# B&R Automation Studio project ksuTCPExample
Automation Studio 4.9

## Configuration Config1

CPU X20CP1586, AutomationRuntime C4.92, Build 4.1.2, Vc V4.72.5

### Task classes (Cpu.sw)
```
Cyclic#8:
  Client <- TCPComms.Client.prg
  Server <- TCPComms.Server.prg [disabled]
Libraries: AsTCP, runtime, BRSE_JSON, astime, sys_lib, AsBrStr, standard, asstring, Queue
```

### Hardware
```
X20CP1586 : X20CP1586 v1.10.0.0
  Connector IF2:
    ActivateDevice = 1
  ConfigurationID = ksuTCPExample_Config1
  Simulation = 1
  VolatileGlobalPvSize = 210000
  FileDevice1
  FileDeviceName1 = USER
  FileDevicePath1 = USER_PATH
```

## Logical view

Binary libraries used (declarations not repeated): operator, runtime, astime, AsIecCon, AsTCP, sys_lib, AsBrStr, standard, asstring

### Global.typ - Global data types
```iecst
TYPE
	MessageToEZ3_typ : 	STRUCT
		Move_Command : STRING[20];
		Parameter_One : STRING[20];
		Parameter_Two : STRING[20];
		Battery_Subscribe : BOOL;
	END_STRUCT;
END_TYPE
```

### Global.var - Global variables
```iecst
VAR
	gSendQueue : FifoQueue_typ;
	gMessageToEZ3 : MessageToEZ3_typ;
END_VAR
```

### Package Logical/Libraries - Global libraries

### Library Logical/Libraries/BRSE_JSON (ANSIC, version 1.00.1) - A new source library
Depends on: sys_lib, astime, AsBrStr

#### BRSE_JSON.fun - Exported functions and function blocks
```iecst
(********************************************************************
 * COPYRIGHT -- B&R
 ********************************************************************
 * Library: Library
 * File: Library.fun
 * Author: Florian Damerow
 * Created: March 09, 2011
 ********************************************************************
 * Functions and function blocks of library Library
 ********************************************************************)

FUNCTION_BLOCK JSON_Parse (*parses a JSON message and writes the content to the structure on the PLC*)
	VAR_INPUT
		pMessage : REFERENCE TO UDINT; (*Pointer to the JSON Message (String)*)
		pDebug : REFERENCE TO UDINT; (*Pointer Debug Buffer (String)*)
		pVariablesNotFound : REFERENCE TO UDINT; (*Pointer Buffer of VariablesNotFound (String)*)
		SizeVariablesNotFound : UDINT; (*size of the VariablesNotFound Buffer*)
		SizeDebug : UDINT; (*size of the Debug Buffer*)
	END_VAR
	VAR_OUTPUT
		ErrorInfo : UINT;
	END_VAR
	VAR
		parselevel : USINT;
		pvIndex : ARRAY[0..MAX_STRUCT_DEPTH_Parse] OF INT;
		Buffer : STRING[80];
		parsestateold : USINT;
		parsestate : USINT;
		pvName : ARRAY[0..MAX_STRUCT_DEPTH_Parse] OF STRING[64];
		isArray : ARRAY[0..MAX_STRUCT_DEPTH_Parse] OF BOOL;
		fullName : STRING[MAX_STRUCT_NAME_LENGTH_Parse];
		j : UINT;
	END_VAR
END_FUNCTION_BLOCK

FUNCTION_BLOCK JSON_Stringify (*converts a PV variable and the whole structure into a JSON Object using PV_ninfo*)
	VAR_INPUT
		pStName : REFERENCE TO UDINT; (*address to variable name (STRING)*)
	END_VAR
	VAR_OUTPUT
		Status : UINT; (*address to status-variable 0=not done; 1=done; 2=error*)
		Output : STRING[MAX_OUTPUT_LENGTH_Stringify]; (*Output contains the content of one step*)
	END_VAR
	VAR
		tmpStruct : STRING[MAX_OUTPUT_LENGTH_Stringify];
		pvName : ARRAY[0..MAX_STRUCT_DEPTH_Stringify] OF STRING[100];
		j : UDINT;
		pvIndex : ARRAY[0..MAX_STRUCT_DEPTH_Stringify] OF UINT;
		TaskDoc : TaskDoc1_typ;
		pvType : UDINT;
		pvLength : UDINT;
		arrMem : ARRAY[0..MAX_STRUCT_DEPTH_Stringify] OF UINT;
		pvStructMembers : ARRAY[0..MAX_STRUCT_DEPTH_Stringify] OF UINT;
		tmpValue : STRING[MAX_OUTPUT_LENGTH_Stringify];
		Buffer : STRING[MAX_OUTPUT_LENGTH_Stringify];
		i : DINT;
		pvLevel : DINT;
		tmpDepth : STRING[MAX_OUTPUT_LENGTH_Stringify];
		state : USINT;
		pvContinue : BOOL;
		pvSearchComplete : BOOL;
		data_len : UDINT;
		isArray : ARRAY[0..MAX_STRUCT_DEPTH_Stringify] OF BOOL;
		arrIndex : UINT;
		pv_adresse : UDINT;
	END_VAR
END_FUNCTION_BLOCK
```

#### BRSE_JSON.c
```c
/*! \file BRSE_JSON.c */
/********************************************************************
 * COPYRIGHT -- B&R
 ********************************************************************
 * Library: BRSE_JSON
 * File: BRSE_JSON.c
 * Author: Florian Damerow
 * Created: March 09, 2011
 *******************************************************************/

#include <bur/plctypes.h>
#include "BRSE_JSON.h"
#include <AsBrStr.h>
#include <string.h>
#include "BRSE_JSON_Main.h"
STRING tmpVal[80];

UDINT ValToString(UDINT pv_adresse, UINT pvType){
	switch (pvType) {
		case 1: {
				BOOL *var = (BOOL *)pv_adresse;
				brsitoa((BOOL)*var,(UDINT)&tmpVal);
				break;
				}
		case 2: {
				SINT *var = (SINT *)pv_adresse;
				brsitoa((SINT)*var,(UDINT)&tmpVal);
				break;
				}
		case 3: {
				INT *var = (INT *)pv_adresse;
				brsitoa((INT)*var,(UDINT)&tmpVal);
				break;
				}
		case 4: {
				DINT *var = (DINT *)pv_adresse;
				brsitoa((DINT)*var,(UDINT)&tmpVal);
				break;
				}
		case 5: {
				USINT *var = (USINT *)pv_adresse;
				brsitoa((USINT)*var,(UDINT)&tmpVal);
				break;
				}
		case 6: {
				UINT *var = (UINT *)pv_adresse;
				brsitoa((UINT)*var,(UDINT)&tmpVal);
				break;
				}
		case 7: {
				UDINT *var = (UDINT *)pv_adresse;
				brsitoa((UDINT)*var,(UDINT)&tmpVal);
				break;
				}
		case 8: {
				REAL *var = (REAL *)pv_adresse;
				brsftoa((REAL)*var,(UDINT)&tmpVal);
				break;
				}
		case 9: {
				STRING *var = (STRING *)pv_adresse;
				STRING *tmpBuffer = (STRING *)&tmpVal;
				strcpy(tmpVal,"\"");
				tmpBuffer++;
				strncpy(tmpBuffer,var,(sizeof(tmpVal)-3));
				strcat(tmpVal,"\"");
				break;
				}
		case 11:{
				DINT *var = (DINT *)pv_adresse;
				STRING *tmpBuffer = (STRING *)&tmpVal;
				strcpy(tmpVal,"\"");
				tmpBuffer++;
				brsitoa((DINT)*var,(UDINT)tmpBuffer);
				strcat(tmpVal,"\"");
				break;
				}
		case 12:{
				DINT *var = (DINT *)pv_adresse;
				STRING *tmpBuffer = (STRING *)&tmpVal;
				strcpy(tmpVal,"\"");
				tmpBuffer++;
				brsitoa((DINT)*var,(UDINT)tmpBuffer);
				strcat(tmpVal,"\"");
				break;
				}
		case 14:{
				LREAL *var = (LREAL *)pv_adresse;
				brsftoa((LREAL)*var,(UDINT)&tmpVal);
				break;
			}
		/*case 11:{
				TIME *var = pv_adresse;
				STRING *ptmpValue = &tmpValue;
				strcpy(ptmpValue,"\\/Date(");
				ptmpValue = ptmpValue + 7;
				itoa((DINT)*var,ptmpValue);
				strcat(ptmpValue,")\\/");
				break;
				}
		case 11:{
				DATE_AND_TIME *var = pv_adresse;
				BRSE_DTF_DateTimeFormat_typ format;
				UDINT error;
				error = BRSE_DTF_CreateFormat("YYYY-MM-DD-hh:mm:ss", &format);
				if(error == 0){
					BRSE_DTF_DTToString((DATE_AND_TIME)*var, &format, tmpValue);
				}
				break;
				}
		case 12:{
				TIME *var = pv_adresse;
				STRING *ptmpValue = &tmpValue;
				strcpy(ptmpValue,"\\/Time(");
				ptmpValue = ptmpValue + 7;
				itoa((DINT)*var,ptmpValue);
				strcat(ptmpValue,")\\/");
				break;
				}*/
		default: strcpy(tmpVal,"null");
				 break;
	}
	return (UDINT)tmpVal;
}

/*! \interface JSON_Parse
	\brief parses a JSON message and writes the content to the structure on the PLC

	This function block parses the JSON message and writes the content to the structure on the PLC using PV_xgetadr.\n
	The structure must exist.\n
	\n
	It is possible to parse a long JSON message in several pieces. The message can be split at every point.\n
	It is only possible to parse JSON Objects '{name:content}' \n
	arrays or non objects are NOT supported e.g. '[name:content, name2:content2]' or 'name:content' \n
	\n
	The maximal possible struture name is defined in MAX_STRUCT_NAME_LENGTH_Parse. \n
	That means the whole name e.g. 'Structure.Outer[1].Inner.Test' is limited. \n
	\n
	Entering an object will result in going up with the level by 1 \n
	Entering an array will result in going up with the level by 1 \n
	Entering an struct array will result in going up with the level by 2 \n
	\n
	If pDebug != 0 the whole message will be written there. This will be done with the state for every character.\n
	If pDebug = 0 no Debugging will be performed by the system.\n

	If pVariablesNotFound != 0 all Variables found in the Message, but could not be written on the system are listed here.
	They are represented in a JSON array e.g. '["var1","var2"]'.\n
	If pVariablesNotFound = 0 no output will performed wen variables could not be written.\n
	\n
	The funktion block will be stopped when an error accured.\n
	The function block will not be stopped when a warning accures.\n
	\par Errors:\n
	\arg 1001	invalid JSON in parsestate 0
	\arg 1002	invalid JSON in parsestate 1
	\arg 1003	invalid JSON in parsestate 3
	\arg 1004	invalid JSON in parsestate 4
	\arg 1005	invalid JSON in parsestate 6
	\arg 1006	invalid JSON in parsestate 7
	\arg 1007	Structure depth is deeper than MAX_STRUCT_DEPTH_Parse

	\par Warnings:\n
	\arg 3001	data type not supported
	\arg 3002	variable not found

	\par General: \n
	\arg 2001	parsing so far successful, but end of JSON message net reached yet
	\arg 0		successfuly finished parsing

	\param[in] pMessage Pointer to the JSON Message (String)
	\param[in] pDebug Pointer Debug Buffer (String)
	\param[in] SizeDebug size of the Debug Buffer
	\param[in] pVariablesNotFound Pointer Buffer of VariablesNotFound (String)
	\param[in] SizeVariablesNotFound size of the VariablesNotFound Buffer

	\param[out] ErrorInfo contains the Error/Warning/General Codes.

*/

void JSON_Parse(struct JSON_Parse* inst)
{
	STRING *message = (STRING *)inst->pMessage;
	STRING *pBuff = (STRING *)inst->pMessage;
	UDINT pBuffOld = 0;
	inst->ErrorInfo = 0;
	while((UDINT)pBuff<((UDINT)message+strlen(message)) && (inst->ErrorInfo < 1000 || inst->ErrorInfo >=2000)){
		switch(inst->parsestate){
			case 0:
				if(*pBuff == '{'){
					inst->parsestate = 1;
					inst->parselevel++;
					pBuff++;
					if(inst->pVariablesNotFound != 0 && inst->SizeVariablesNotFound > 2){
						strcpy((STRING *)inst->pVariablesNotFound,"[");
					}
				}
				else if(*pBuff == ' '){
					pBuff++;
				}
				else{
					inst->ErrorInfo = 1001; /*invalid JSON*/
					return;
				}
				break;

			case 1:
				if(*pBuff == '"'){
					inst->parsestate = 2;
					pBuff++;
				}
				else if(*pBuff == ' '){
					pBuff++;
				}
				else{
					inst->ErrorInfo = 1002; /*invalid JSON*/
					return;
				}
				break;

			case 2:
				if(*pBuff != '"'){
					inst->pvName[inst->parselevel][inst->j] = *pBuff;
					inst->j++;
					pBuff++;
				}
				else {
					inst->pvName[inst->parselevel][inst->j] = '\0';
					inst->j = 0;
					inst->parsestate = 3;
					pBuff++;
				}
				break;

			case 3:
				if(*pBuff == ':'){
					inst->parsestate = 4;
					pBuff++;
				}
				else if(*pBuff == ' '){
					pBuff++;
				}
				else{
					inst->ErrorInfo = 1003; /*invalid JSON*/
					return;
				}
				break;

			case 4:
				if(*pBuff == '{'){
					inst->parsestate = 1;
					inst->parselevel++;
					pBuff++;
				}
				else if(*pBuff == '['){
					/*strcat(inst->pvName[inst->parselevel],"[");
					strcat(inst->pvName[inst->parselevel],"0");
					strcat(inst->pvName[inst->parselevel],"]");*/
					inst->isArray[inst->parselevel] = 1;
					inst->parselevel++;
					pBuff++;
				}
				else if(*pBuff == '\"'){
					inst->Buffer[inst->j] = *pBuff;
					pBuff++;
					inst->j++;
					inst->parsestate = 41;
				}
				else if(*pBuff != '{' && *pBuff != ' ' && *pBuff != '['){ /*maybe better to check for " or - or number*/
					inst->parsestate = 5;
				}
				else if(*pBuff == ' '){
					pBuff++;
				}
				else{
					inst->ErrorInfo = 1004; /*invalid JSON*/
					return;
				}
				break;

			case 41: /* is in String */
				if(*pBuff == '\"'){
					inst->Buffer[inst->j] = *pBuff;
					inst->j++;
					inst->Buffer[inst->j] = '\0';
					inst->j=0;
					pBuff++;
					inst->parsestate = 51;
				}
				else if(*pBuff == '\\'){
					inst->Buffer[inst->j] = *pBuff;
					inst->j++;
					pBuff++;
					inst->Buffer[inst->j] = *pBuff;
					inst->j++;
					pBuff++;
				}
				else{
					inst->Buffer[inst->j] = *pBuff;
					inst->j++;
					pBuff++;
				}
				break;

			case 5:
				if(*pBuff != '}' && *pBuff != ' ' && *pBuff != ',' && *pBuff != ']'){
					inst->Buffer[inst->j] = *pBuff;
					inst->j++;
					pBuff++;
				}
				else{
					inst->Buffer[inst->j] = '\0';
					inst->j=0;
					inst->parsestate = 51;
				}
				break;

			case 51: /*write variable*/
				memset((UDINT *)(inst->fullName),0,sizeof(inst->fullName));
				{
					UINT i = 1;
					UDINT adresse;
					UDINT datalen;
					UDINT pvType;
					UDINT pvLength;
					UINT pvStructMembers;
					STRING tmpStr[5];
					while(i <= inst->parselevel && (sizeof(inst->fullName)-strlen(inst->fullName)-7) > strlen(inst->pvName[i])){
						strcat(inst->fullName,inst->pvName[i]);
						if(inst->isArray[i] == 1){
							strcat(inst->fullName,"[");
							brsitoa(inst->pvIndex[i],(UDINT)&tmpStr);
							strcat(inst->fullName,tmpStr);
							strcat(inst->fullName,"]");
						}
						if(i < inst->parselevel && inst->isArray[i] == 0){
							strcat(inst->fullName,".");
						}
						i++;
					}
					inst->ErrorInfo = PV_ninfo((STRING *)&inst->fullName, &pvType, &pvLength, &pvStructMembers);
					if(inst->ErrorInfo == 0){
						inst->ErrorInfo = PV_xgetadr((STRING *)&inst->fullName, &adresse, &datalen);
					}
					else{
						inst->ErrorInfo = 3002; /* variable not found */
					}
					if(inst->ErrorInfo == 0){
						STRING *Buffer = (STRING *)&inst->Buffer;
						if(*Buffer == '\"'){
							Buffer++;
							if(inst->Buffer[strlen(Buffer)] == '\"'){
								inst->Buffer[strlen(Buffer)] = '\0';
							}
						}
						if(strstr(inst->Buffer,"null") == 0){
							switch(pvType){
								case 0:{
									DINT *adr = (DINT *)adresse;
									*adr = (DINT)brsatoi((UDINT)Buffer);
									break;
									}
								case 1:{
									BOOL *adr = (BOOL *)adresse;
									if(brsatoi((UDINT)Buffer) != 0){
										*adr = 1;
									}
									else{
										*adr = 0;
									}
									break;
									}
								case 2:{
									SINT *adr = (SINT *)adresse;
									*adr = (SINT)brsatoi((UDINT)Buffer);
									break;
									}
								case 3:{
									INT *adr = (INT *)adresse;
									*adr = (INT)brsatoi((UDINT)Buffer);
									break;
									}
								case 4:{
									DINT *adr = (DINT *)adresse;
									*adr = (DINT)brsatoi((UDINT)Buffer);
									break;
									}
								case 5:{
									USINT *adr = (USINT *)adresse;
									*adr = (USINT)brsatoi((UDINT)Buffer);
									break;
									}
								case 6:{
									UINT *adr = (UINT *)adresse;
									*adr = (UINT)brsatoi((UDINT)Buffer);
									break;
									}
								case 7:{
									UDINT *adr = (UDINT *)adresse;
									*adr = (UDINT)brsatoi((UDINT)Buffer);
									break;
									}
								case 8:{
									REAL *adr = (REAL *)adresse;
									*adr = (REAL)brsatof((UDINT)Buffer);
									break;
									}
								case 9:{
									STRING *adr = (STRING *)adresse;
									strncpy(adr, Buffer, pvLength-1);
									break;
									}
								case 11:{
									DINT *adr = (DINT *)adresse;
									*adr = (DINT)brsatoi((UDINT)Buffer);
									break;
									}
								case 12:{
									DINT *adr = (DINT *)adresse;
									*adr = (DINT)brsatoi((UDINT)Buffer);
									break;
									}
								case 14:{
										LREAL *adr = (LREAL *)adresse;
										*adr = (LREAL)brsatof((UDINT)Buffer);
										break;
									}
								/*case 11:{
									DINT *adr = adresse;
									STRING *Buffer = &inst->Buffer;
									Buffer = strstr(inst->Buffer,")\\/");
									if(Buffer != 0){
										*Buffer = '\0';
										Buffer = strstr(inst->Buffer,"\\/Date(");
										if(Buffer != 0){
											Buffer = Buffer + 7;
										}
									}
									*adr = (DINT)atoi(Buffer);
									break;
									}
								case 12:{
									DINT *adr = adresse;
									STRING *Buffer = &inst->Buffer;
									Buffer = strstr(inst->Buffer,")\\/");
									if(Buffer != 0){
										*Buffer = '\0';
										Buffer = strstr(inst->Buffer,"\\/Time(");
										if(Buffer != 0){
											Buffer = Buffer + 7;
										}
									}
									*adr = (DINT)atoi(Buffer);
									break;
									}*/

								default:{
									inst->ErrorInfo = 3001;
									break;
									}
							}
						}
					}
					else{
						inst->ErrorInfo = 3002; /* variable not found */
						if(inst->pVariablesNotFound != 0 && inst->SizeVariablesNotFound != 0){
							if((inst->SizeVariablesNotFound - strlen((STRING *)inst->pVariablesNotFound)-2) > strlen(inst->fullName)+3){
								if(strlen((STRING *)inst->pVariablesNotFound) > 2){
									strcat((STRING *)inst->pVariablesNotFound,",");
								}
								strcat((STRING *)inst->pVariablesNotFound,"\"");
								strcat((STRING *)inst->pVariablesNotFound,inst->fullName);
								strcat((STRING *)inst->pVariablesNotFound,"\"");
							}
						}
					}
					if(*pBuff == ',' && inst->isArray[inst->parselevel-1] == 1){
						pBuff++;
						inst->pvIndex[inst->parselevel-1]++;
						inst->parsestate = 4;
					}
					else{
						inst->parsestate = 6;
					}
				}
				break;

			case 6:
				if(*pBuff == '}'){
					inst->parsestate = 6;
					inst->pvIndex[inst->parselevel-1] = 0;
					inst->parselevel--;
					pBuff++;
				}
				else if(*pBuff == ']'){
					inst->parsestate = 6;
					inst->pvIndex[inst->parselevel-1] = 0;
					inst->parselevel--;
					inst->isArray[inst->parselevel] = 0;
					pBuff++;
				}
				else if(*pBuff == ','){
					inst->parsestate = 7;
					inst->pvIndex[inst->parselevel-1]++;
					pBuff++;
				}
				else if(*pBuff == ' '){
					pBuff++;
				}
				else{
					inst->ErrorInfo = 1005; /*invalid JSON*/
					return;
				}
				break;

			case 7:
				if(*pBuff == '{'){
					inst->parselevel++;
					inst->parsestate = 1;
					pBuff++;
				}
				else if(*pBuff == '\"'){
					inst->parsestate = 1;
				}
				else if(*pBuff == ' '){
					pBuff++;
				}
				else{
					inst->ErrorInfo = 1006; /*invalid JSON*/
					return;
				}
		}

		/* DEBUGGING */
		if(inst->pDebug != 0){
			if(pBuffOld != (UDINT)pBuff){
				STRING BUFFER2[4];
				STRING BUFFER3[2];
				if((inst->SizeDebug - strlen((STRING *)inst->pDebug) - 1) > 7){
					if(inst->parsestateold != inst->parsestate){
						inst->parsestateold = inst->parsestate;
						brsitoa((DINT)inst->parsestate,(UDINT)&BUFFER2);
						strcat((STRING *)inst->pDebug,"(");
						strcat((STRING *)inst->pDebug,BUFFER2);
						strcat((STRING *)inst->pDebug,")");
					}
					BUFFER3[0] = *pBuff;
					BUFFER3[1] = 0;
					strcat((STRING *)inst->pDebug,BUFFER3);
				}
			}
			pBuffOld = (UDINT)pBuff;
		}
	}
	/* Error Handling */
	if(inst->parselevel > MAX_STRUCT_DEPTH_Parse){
		inst->ErrorInfo = 1007;
	}
	if(inst->ErrorInfo >= 1000 && inst->ErrorInfo  < 2000){
		inst->parselevel = 0;
		inst->parsestate = 0;
		memset(inst->pvIndex,0,sizeof(inst->pvIndex));
		memset(inst->pvName,0,sizeof(inst->pvName));
	}
	else if(inst->parselevel != 0){
		inst->ErrorInfo = 2001; /*not done*/
	}
	else{
		if(inst->pVariablesNotFound != 0){
			strcat((STRING *)inst->pVariablesNotFound,"]");
		}
		inst->parsestate = 0;
	}
}

/*! \interface JSON_Stringify
	\brief converts a PV variable and the whole structure into a JSON Object using PV_ninfo.

	This function block converts the whole structure of a PV variable into a JSON Object using PV_ninfo. \n
	The variable name should be the same as using the PV_ninfo function. By that it is possible to access any kind of PV variables.\n
	The output is always a JSON object. e.g. '{"varname": ... }' \n
	\n
	The function block has to be run several times until the Status = 1. \n
	Every time the function block is called it creates the JSON output for one new variable inside the Structure. \n
	If the variable in the structure is an array of a non object type the whole array will be created in Output.\n
	\n
	The maximum Output length is defined by MAX_OUTPUT_LENGTH_Stringify.\n
	The maximum Value of a nun array, non structure variable is 80. So Strings are only supported up the 80 characters.\n

	\par Status Codes:\n
	\arg 1001 Variable not found
	\arg 1002 Variable value too long
	\arg 1 singify process completed
	\arg 0 singify process not completet yet - run again

	\param[in] pStName Pointer to the requested variable name

	\param[out] Status returns the Status codes
	\param[out] Output contains the content of one step

*/
void JSON_Stringify(struct JSON_Stringify* inst)
{
	STRING *pBuff = 0;
	STRING strBuff[20];
	inst->TaskDoc.Input.StructDepth = MAX_STRUCT_DEPTH_Stringify;
	/*gather information of the structure item*/
	memset(inst->tmpStruct,0,sizeof(inst->tmpStruct));
	strcpy(inst->tmpStruct,(STRING *)inst->pStName);

	strcat(inst->tmpStruct, inst->pvName[0]);
	for( inst->i = 1; inst->i <= inst->pvLevel; inst->i++ ){
		if(inst->isArray[inst->i-1] == 0){
			strcat(inst->tmpStruct, ".");
			strcat(inst->tmpStruct, inst->pvName[inst->i]);
		}
		else{
			inst->isArray[inst->pvLevel] = 1;
			strcat(inst->tmpStruct,"[");
			brsitoa(inst->pvIndex[inst->i-1],(UDINT)&strBuff);
			strcat(inst->tmpStruct,strBuff);
			strcat(inst->tmpStruct,"]");
		}
	}
	/*Search in PV-list*/
	inst->TaskDoc.Output.StatusInfo = PV_ninfo((STRING *)&inst->tmpStruct, &inst->pvType, &inst->pvLength, &inst->pvStructMembers[inst->pvLevel]);
	if(inst->pvType == 0){
		STRING name[80];
		inst->TaskDoc.Output.StatusSearch = PV_item((STRING *)&inst->tmpStruct, 0, (STRING *)&name);
		if(inst->TaskDoc.Output.StatusSearch != 0){
			inst->pvType = 4;
			inst->pvStructMembers[inst->pvLevel] = 1;
			inst->TaskDoc.Output.StatusSearch = 0;
		}
	}
	if(inst->pvType == 15){
		inst->isArray[inst->pvLevel] = 1;
		strcat(inst->tmpStruct,"[");
		brsitoa(inst->pvIndex[inst->pvLevel],(UDINT)&strBuff);
		strcat(inst->tmpStruct,strBuff);
		strcat(inst->tmpStruct,"]");
		inst->pvLevel = inst->pvLevel + 1;
		inst->TaskDoc.Output.StatusInfo = PV_ninfo((STRING *)&inst->tmpStruct, &inst->pvType, &inst->pvLength, &inst->pvStructMembers[inst->pvLevel]);
	}
	else{
		inst->isArray[inst->pvLevel] = 0;
	}
	if( inst->TaskDoc.Output.StatusInfo == 0 ){
		inst->TaskDoc.Output.StatusInfo = PV_xgetadr((STRING *)&inst->tmpStruct,&inst->pv_adresse,&inst->data_len);
	}
	if( inst->TaskDoc.Output.StatusInfo == 0 ){
	/*variable was found*/
		STRING *ValToStr;
		UDINT Size=0;
		memset(inst->tmpValue,0,sizeof(inst->tmpValue));
		if(inst->pvStructMembers[inst->pvLevel]>1){
			strcat(inst->tmpValue,"[");
		}
		ValToStr = (STRING *)ValToString(inst->pv_adresse, inst->pvType);
		if((sizeof(inst->tmpValue)-strlen(inst->tmpValue)-2) > strlen(ValToStr)){
			strcat(inst->tmpValue, ValToStr);
		}
		inst->arrIndex = 1;
		Size = (UDINT)(inst->data_len/inst->pvStructMembers[inst->pvLevel]);
		pBuff = (STRING *)((UDINT)inst->pv_adresse+Size);
		/*build array output */
		while(inst->arrIndex < inst->pvStructMembers[inst->pvLevel]){
			ValToStr = (STRING *)ValToString((UDINT)pBuff, inst->pvType);
			if((sizeof(inst->tmpValue)-strlen(inst->tmpValue)-2) <= strlen(ValToStr)){
				inst->Status = 1002; /*Variable Value too long*/
				return;
			}
			strcat(inst->tmpValue, ",");
			strcat(inst->tmpValue, ValToStr);
			pBuff = pBuff+Size;
			inst->arrIndex++;
		}
		if(inst->pvStructMembers[inst->pvLevel]>1){
			strcat(inst->tmpValue,"]");
		}

		/*get inner variable name*/
		pBuff = (inst->tmpStruct)+strlen(inst->tmpStruct);
		while((UDINT)pBuff >= (UDINT)&(inst->tmpStruct) && *pBuff != '.'){
			pBuff--;
		}
		pBuff++;
		/*create JSON output*/
		memset(inst->Output,0,sizeof(inst->Output));
		if((43+strlen(inst->tmpValue)) > sizeof(inst->Output)){
			inst->Status = 1002; /*Variable Value too long*/
			return;
		}
		if(!(inst->isArray[inst->pvLevel-1] == 1 && inst->pvIndex[inst->pvLevel-1] > 0)){
			if((inst->pvLevel == 0 && inst->pvIndex[0] == 0) || (inst->isArray[inst->pvLevel-1] == 1 && (inst->pvLevel-1) == 0) ){
				strcat(inst->Output, "{");

			}
			strcat(inst->Output, "\"");
			if( inst->pvLevel == 0){
				strcat(inst->Output, (STRING *)inst->pStName);
			}
			else if(inst->isArray[inst->pvLevel-1] == 1){
				if((inst->pvLevel-1) > 0){
					strcat(inst->Output, inst->pvName[inst->pvLevel-1]);
				}
				else{
					strcat(inst->Output, (STRING *)inst->pStName);
				}
			}else{
				strcat(inst->Output, inst->pvName[inst->pvLevel]);
			}
			strcat(inst->Output, "\":");
			if(inst->isArray[inst->pvLevel-1]){
				strcat(inst->Output, "[");
			}
		}
		if( inst->pvType == 0 ){
			strcat(inst->Output, "{");
		}
		if( inst->pvType != 0 && inst->pvType != 15 ){
			strcat(inst->Output, inst->tmpValue);
		}

		inst->pvSearchComplete = 0;

		if( (inst->pvType == 0) && (inst->pvLevel < (inst->TaskDoc.Input.StructDepth-1)) ){
			/*variable is a structure and its ok to go look inside it*/
			/*ok. proceed to next level.*/
			inst->TaskDoc.Output.StatusSearch = PV_item((STRING *)&inst->tmpStruct, inst->pvIndex[inst->pvLevel], (STRING *)&inst->pvName[inst->pvLevel+1]);
			inst->pvLevel = inst->pvLevel + 1;
		}
		else if( (inst->pvLevel > 0) || (inst->pvLevel==0 && inst->pvIndex[inst->pvLevel] < (inst->pvStructMembers[inst->pvLevel]))){ /*..in case its 0 we have a problem*/
		/*variable is a basic datatype*/
			do{
				inst->pvContinue = 0;
				if( inst->isArray[inst->pvLevel-1] == 1){
					if( inst->pvIndex[inst->pvLevel-1] < (inst->pvStructMembers[inst->pvLevel-1]-1)){
						/*ok. take the next item in prior structure*/
						inst->pvIndex[inst->pvLevel-1] = inst->pvIndex[inst->pvLevel-1] + 1;
						inst->pvLevel = inst->pvLevel - 1;
						strcat(inst->Output, ",");
						break; /*..from loop*/
					}
					else{
						strcat(inst->Output, "]");
						inst->pvLevel = inst->pvLevel - 1;
						inst->pvIndex[inst->pvLevel] = 0;
						if( inst->pvLevel > 0 ){
							inst->pvContinue = 1;
						}else{
							inst->pvSearchComplete = 1;
							strcat(inst->Output, "}");
							break;
						}
					}
				}
				else{
					if( inst->pvIndex[inst->pvLevel-1] < (inst->pvStructMembers[inst->pvLevel-1]-1)){
						/*ok. take the next item in prior structure*/
						inst->pvIndex[inst->pvLevel-1] = inst->pvIndex[inst->pvLevel-1] + 1;
						strcat(inst->Output, ",");
						break; /*..from loop*/
					}else{
						/*continue looking in the prior structure if the index is smaller members*/
						inst->pvLevel = inst->pvLevel - 1;
						if(inst->pvLevel>=0){
							strcat(inst->Output, "}");
						}
						inst->pvIndex[inst->pvLevel] = 0; /*this one is used the nest time a structure is found on this level*/
						if( inst->pvLevel > 0 ){
							inst->pvContinue = 1;
						}else{
							inst->pvSearchComplete = 1;
							strcat(inst->Output, "}");
							break;
						}
					}
				}
			}
			while(inst->pvContinue != 0);

			/*look after following member in prior structure*/
			if( inst->pvLevel > 0 ){
				strcpy(inst->tmpStruct,(STRING *)inst->pStName);

				strcat(inst->tmpStruct, inst->pvName[0]);
				for( inst->i = 1; inst->i <= (inst->pvLevel-1); inst->i++ ){
					if(strlen(inst->pvName[inst->i]) != 0){
						strcat(inst->tmpStruct, ".");
						strcat(inst->tmpStruct, inst->pvName[inst->i]);
					}
				}
				/*ok. get the next variable*/
				inst->TaskDoc.Output.StatusSearch = PV_item((STRING *)&inst->tmpStruct, inst->pvIndex[inst->pvLevel-1], (STRING *)&inst->pvName[inst->pvLevel]);
			}else if((inst->pvLevel==0 && inst->pvIndex[inst->pvLevel] == (inst->pvStructMembers[inst->pvLevel]))){
				/*no more items in top structure*/
				inst->pvSearchComplete = 1;
			}
		}else{
			inst->pvSearchComplete = 1;
		}
		if(inst->pvSearchComplete == 1){
			inst->Status = 1;
		}else{
			inst->Status = 0;
		}
	}else{
		 inst->Status = 1001; /*variable not found*/
	}
}
```

#### BRSE_JSON.typ - Exported data types
```iecst
(********************************************************************
 * COPYRIGHT -- B&R
 ********************************************************************
 * Library: BRSE_JSON
 * File: BRSE_JSON.typ
 * Author: Florian Damerow
 * Created: March 09, 2011
 ********************************************************************
 * Data types of library BRSE_JSON
 ********************************************************************)

TYPE
	TaskDoc1_typ : 	STRUCT
		Output : Output1_typ;
		Input : Input1_typ;
		State : USINT;
	END_STRUCT;
	Input1_typ : 	STRUCT
		StructDepth : DINT;
	END_STRUCT;
	Output1_typ : 	STRUCT
		StatusGet : UINT;
		StatusInfo : UINT;
		StatusSearch : UINT;
	END_STRUCT;
END_TYPE
```

#### BRSE_JSON_Main.h
```c
/*! \file BRSE_JSON_Main.h */
/*!
	\mainpage BRSE_JSON

	\section Introduction
	\brief This library provides the ability to use JSON to write and read variables using normal ASCII string communication.

	\section Usage
	The library contains two function blocks \ref JSON_Parse and \ref JSON_Stringify.

	\ref JSON_Parse takes a JSON string created by \ref JSON_Stringify and interprets it.
	It searches for the variables and updates their values on the PLC.

	\ref JSON_Stringify takes an address to a string containing a variable or structure name and creates a JSON string.
	The JSON string contains all the necessary data about the structure or variable so that a parser can reconstruct it.
	It uses a basic JSON structure: {name:content}

	An example of a string is the following:

	{"PV_var1":[{"Outer1":[{"Middle2":"1234","Middle1":[{"Inner1":"90","Inner2":"22","Inner3":"33"}]}]"Outer2":"567"}]}

	The JSON string describes the following structure:

	PV_var1 \n
	...=>Outer1 \n
	......=>Middle2 1234 \n
	......=>Middle1 \n
	.........=>Inner1 90 \n
	.........=>Inner2 22 \n
	.........=>Inner3 33 \n
	...=>Outer2 567
*/

#include "BRSE_JSON.h"
#include <asstring.h>
#include <string.h> /*this will override the asstring functions*/
```

#### BRSE_JSON.var - Exported constants
```iecst
(********************************************************************
 * COPYRIGHT -- B&R
 ********************************************************************
 * Library: BRSE_JSON
 * File: BRSE_JSON.var
 * Author: Florian Damerow
 * Created: April 05, 2011
 ********************************************************************
 * Constants of library BRSE_JSON
 ********************************************************************)
VAR CONSTANT
	MAX_STRUCT_NAME_LENGTH_Parse : USINT := 200;
	MAX_STRUCT_DEPTH_Stringify : USINT := 20;
	MAX_STRUCT_DEPTH_Parse : USINT := 20;
	MAX_OUTPUT_LENGTH_Stringify : UDINT := 20000;
END_VAR
```

#### example.c
```c
/*! \page Example

\section Example Task

This task is used together with the JSON Client (see next section) to read and send data using JSON.
Making it possible to read/write variables and create files through a normal webbrowser.
\arg Global Types
\code
TYPE
	New_typ1 : 	STRUCT
		Middle2 : UINT;
		Middle1 : ARRAY[0..1] OF New_typ;
	END_STRUCT;
	New_typ : 	STRUCT
		Inner1 : ARRAY[0..10] OF SINT;
		Inner2 : UINT;
		Inner3 : DATE_AND_TIME;
		Inner5 : ARRAY[0..2] OF STRING[20];
	END_STRUCT;
	PV_var_typ : 	STRUCT
		Outer1 : ARRAY[0..1] OF New_typ1;
		Outer2 : BOOL;
	END_STRUCT;
	ParameterMachineDayTank_typ : 	STRUCT
		ChemicalType : USINT;
	END_STRUCT;
	ParameterMachine_typ : 	STRUCT
		DayTank : ARRAY[0..MAX_NUMBER_OF_DAYTANKS_MACHINE] OF ParameterMachineDayTank_typ;
		NumberOfDayTanks : USINT;
	END_STRUCT;
	ParameterMainTank_typ : 	STRUCT
		ChemicalType : USINT; (*Type of chemical tank (0 - 8)*)
		LowLevel : INT; (*Level when not able to run the machine (0 - 100%)*)
		OrderLevel : INT; (*Level when to make an order alarm (0 - 100%)*)
		TimeBeforeCirculation : TIME; (*Time before cirulation is done in a circulating system*)
		CirculationTime : TIME; (*How long are the circulation done*)
		MaxTimeForPump : TIME; (*Maximum time of pump beeing run before alarm*)
	END_STRUCT;
	Parameter_typ : 	STRUCT
		MainTank : ARRAY[0..MAX_NUMBER_OF_MAINTANKS] OF ParameterMainTank_typ;
		Machine : ARRAY[0..MAX_NUMBER_OF_MACHINES] OF ParameterMachine_typ;
		NumberOfMainTanks : USINT;
		NumberOfMachines : USINT;
		SystemType : USINT; (*Circulating or Manifold*)
		SetupDone : BOOL; (*The setup of the machine is done*)
	END_STRUCT;
	MAIN_STATES :
		(
		MAIN_INIT, (*Wait for init*)
		MAIN_AUTO, (*System running*)
		MAIN_STOP, (*System stoped*)
		MAIN_FORCEIO (*Force IO*)
		);
	MainInputCommand_typ : 	STRUCT  (*..documented in the code*)
		Auto : BOOL;
		Stop : BOOL;
		EmergencyStop : BOOL;
		ForceIO : BOOL;
		Reset : BOOL;
	END_STRUCT;
	MainInputAccess_typ : 	STRUCT  (*Adresses to other interfaces which are accessed*)
		OtherInterface : UDINT;
	END_STRUCT;
	MainInput_typ : 	STRUCT
		Command : MainInputCommand_typ;
		Access : MainInputAccess_typ;
	END_STRUCT;
	MainOutputStatus_typ : 	STRUCT  (*..documented in the code*)
		SystemRunning : BOOL;
		SystemStoped : BOOL;
		ForceIOActive : BOOL;
		EmergencyStop : BOOL;
		MaintankLowLevel : BOOL;
		DaytankOverfilled : BOOL;
		PumpRunToLong : BOOL;
		LeakOnMaintank : BOOL;
		HighPressure : BOOL;
		OrderConsumables : BOOL;
	END_STRUCT;
	MainOutput_typ : 	STRUCT
		Status : MainOutputStatus_typ;
		DaytankNumberOverfilled : USINT; (*What is my purpose?*)
		MachineNumberOverfilled : USINT; (*What is my purpose?*)
	END_STRUCT;
	Main_typ : 	STRUCT
		Address : UDINT;
		Input : MainInput_typ;
		Output : MainOutput_typ;
		State : MAIN_STATES;
		SubState : UINT;
	END_STRUCT;
END_TYPE

\endcode

\arg Global Variables
\code

	VAR RETAIN
		PV_var1 : ARRAY[0..2] OF PV_var_typ;
		File_List : FILE_LIST_typ;
		Main : ARRAY[0..MAX_NUMBER_OF_MAINTANKS] OF Main_typ;
		Parameter : Parameter_typ;
	END_VAR
	VAR CONSTANT
		MAX_NUMBER_OF_MAINTANKS : USINT := 4;
		MAX_NUMBER_OF_DAYTANKS_MACHINE : USINT := 3;
		MAX_NUMBER_OF_MACHINES : USINT := 7;
	END_VAR

\endcode

\arg Local Variabels
\code
	VAR RETAIN
		BigBuffer : ARRAY[0..400] OF STRING[50];
		Debug : ARRAY[0..29] OF STRING[50];
		VariablesNotFound : ARRAY[0..29] OF STRING[50];
		StName : STRING[60] := 'Parameter';
		JSON_STRINGIFY_0 : JSON_Stringify;
		JSON_PARSE_0 : JSON_Parse;
		CtrlVar : USINT;
		STATUS : UDINT;
		JSONBuffer : ARRAY[0..99] OF STRING[50];
		notreadrd : UDINT := 0;
		readsize : UDINT := 0;
		pOuter : REFERENCE TO New_typ1;
	END_VAR
\endcode

\arg Init
\code
	PROGRAM _INIT

		(* Make the PV variables accessable *)
		PV_var1[0].Outer1[0].Middle1[0].Inner1[0] := 0;
		Parameter.Machine[0].DayTank[0].ChemicalType := 0;
		Main[0].Input.Access.OtherInterface := 0;
		pOuter ACCESS ADR(PV_var1[0].Outer1[0]);	(* pointer variables can be accessed by "JSON_DEMO:*pOuter" *)

		(* define the output for the Webserver *)
		WEB_INIT();
		WEB_PAGE(ADR('/'));					(* Link to the admin panel *)
		WEB_HTML(ADR('<html><body><h1><font color="orange">B&R SGC Webserver with JSON support</font></h1><br><a href="/admin.br">Admin Panel</a></body></html> '));
		WEB_PAGE(ADR('/read'));
		WEB_HTML(ADR(JSONBuffer)); 			(* response of the Stringify function after reading a variable *)
		WEB_PAGE(ADR('/write'));
		WEB_HTML(ADR(VariablesNotFound)); 	(* the variables that could not be found by the Parse function after writing a variable *)
		WEB_PAGE(ADR('/writetofile'));
		WEB_HTML(ADR(JSONBuffer));			(* {"result":true} for success {"result":false} if writing the file failed *)

		(* try to read the file and parse the content => Variable will be written during startup *)
		notreadrd := 1;
		WHILE notreadrd = 1 DO
			notreadrd := FILE_READ(File_List,ADR('setPVvar1.txt'),readsize);
			IF notreadrd < 2 THEN
				readsize := readsize + strlen(FILE_OUTPUT());
				JSON_PARSE_0.pVariablesNotFound := ADR(VariablesNotFound);
				JSON_PARSE_0.SizeVariablesNotFound := SIZEOF(VariablesNotFound);
				JSON_PARSE_0.pDebug := ADR(Debug);
				JSON_PARSE_0.SizeDebug := SIZEOF(Debug);
				JSON_PARSE_0.pMessage := FILE_OUTPUT();
				JSON_PARSE_0();
			END_IF
		END_WHILE

	END_PROGRAM
\endcode

\arg Cyclic
\code
	PROGRAM _CYCLIC

		STATUS := FILE_WEBSER(BigBuffer[0], SIZEOF(BigBuffer), ADR(CtrlVar),File_List); (* run webserver *)

		IF CtrlVar=1 THEN 												(* stop webserver between read and output process *)
			(* memset to restart the function blocks *)
			memset(ADR(JSON_STRINGIFY_0),0,SIZEOF(JSON_STRINGIFY_0));
			memset(ADR(JSON_PARSE_0),0,SIZEOF(JSON_PARSE_0));
			memset(ADR(JSONBuffer),0,SIZEOF(JSONBuffer));

			IF strcmp(HTTP_URL(),ADR('/write'))=0 THEN					(* start parse/write process when the url '/write' is called *)
				JSON_PARSE_0.pVariablesNotFound := ADR(VariablesNotFound);
				JSON_PARSE_0.SizeVariablesNotFound := SIZEOF(VariablesNotFound);
				JSON_PARSE_0.pDebug := ADR(Debug);
				JSON_PARSE_0.SizeDebug := SIZEOF(Debug);
				JSON_PARSE_0.pMessage := HTTP_POST(ADR(BigBuffer));		(* POST content of the Request is JSON request *)
				JSON_PARSE_0();

			ELSIF strcmp(HTTP_URL(),ADR('/writetofile'))=0 THEN			(* overwrite file with new content if the url 'writetofile' is called *)
				FILE_DELETE(File_List,ADR('setPVvar1.txt'));
				IF FILE_STORE(File_List,ADR('setPVvar1.txt'),HTTP_POST(ADR(BigBuffer)),strlen(HTTP_POST(ADR(BigBuffer)))) = 1 THEN
					strcpy(ADR(JSONBuffer),ADR('{"result":true}'));		(* put response the the Webserver Output *)
				ELSE
					strcpy(ADR(JSONBuffer),ADR('{"result":false}'));
				END_IF

			ELSIF strcmp(HTTP_URL(),ADR('/read'))=0 THEN				(* read and stringify the requested Variable *)
				strcpy(ADR(StName),HTTP_POST(ADR(BigBuffer)));
				JSON_STRINGIFY_0.pStName := ADR(StName);
				WHILE JSON_STRINGIFY_0.Status = 0 DO					(* run stringify until the whole structure is created *)
					JSON_STRINGIFY_0();
					IF (SIZEOF(JSONBuffer)-strlen(ADR(JSONBuffer))-1) > strlen(ADR(JSON_STRINGIFY_0.Output)) THEN
						strcat(ADR(JSONBuffer),ADR(JSON_STRINGIFY_0.Output));
					END_IF
				END_WHILE
			END_IF
			CtrlVar:=0; (* webserver continues with output process *)
		END_IF

	END_PROGRAM
\endcode

\section Example JSON Script
This script shows how JSON data structuring can be used to read and set variables.
The interface is easy to use and shows the user what strings the JSON parser is working with.
\image html SCRIPTOV.jpg
It is possible to select working variable and server IP.
There are three different example structures available. Main and Parameter fakes a process interface which makes the structure easy to relate to.
Ideal for presenting the library.

By selecting METHOD and klicking send different commands can be executed.

READ: Reads the value(s) from the variable(structure). \n
WRITE: Writes the values present in the webbrowser to the CPU. Need to build the output first. \n
WRITE TO FILE: Stores the values to a file on the CPU so that they can be loaded after a restart. Need to build the output first. \n

Requirement: There must be a data object called "CFGDMLIB" which contains a value greater than 3 for the file handling to work.
See the standard library DM_lib for more information. Also, make sure that the runtime version is D2.31 or newer.

Some interresting line of codes for the user is the where the IP and the the working variable is set incase the user whants to use a different standard IP and variable.
\image html STANDARDIPANDVAR.jpg

Create a html file with the following content. Save and run in Internet Explorer. Change the IP to match the CPU.

\code
	<html>
	   <style type="text/css">
		table {font-family: arial; font-size : 10pt;}
		blockquote { margin-top: 0px; margin-bottom: 0px; padding: 0px; }
	   </style>

	    <head>
	        <title>JSON</title>
	        <script type="text/javascript">

	         var responseObject = null;
	         var req = null;
	         var output1 = '';

	function isArray(obj) {
	    //returns true is it is an array
	    if (obj.constructor.toString().indexOf('Array') == -1)
	        return false;
	    else
	        return true;
	}

	function valuesToObject(o,Name) {
	    var type = typeof o
	    var outName = Name;
	    if (type == "object") {
	        for (var key in o) {
	            if(!isArray(o)){
	                if(Name != ''){
	                    outName = Name + "['" + key + "']";
	                }
	                else{
	                    outName = Name + "['" + key + "']";
	                }
	            }
	            else{
	                outName = Name + '[' + key + ']';
	            }
	            valuesToObject(o[key],outName);
	        }
	    }
	    else{
	        var test1 = '\'' + document.getElementById(outName).value + '\'';
	        eval('responseObject' + outName + '=' + test1);
	    }
	}

	function js_traverse(o,Name,lastkey) {
	    var type = typeof o
	    var outName = Name;
	    if (type == "object") {
	        if(!isArray(o))
	            output1 = output1 + '<br>{<blockquote>';
	        for (var key in o) {
	            if(!isArray(o)){
	                output1 = output1 + key;
	                if(Name != ''){
	                    outName = Name + "['" + key + "']";
	                    //outName = Name + '.' + key;
	                }
	                else{
	                    outName = Name + "['" + key + "']";
	                    //outName = Name + key;
	                }
	            }
	            else{
	                if(key != '0'){
	                    output1 = output1 + lastkey + '[' + key + ']';
	                }
	                else{
	                    output1 = output1 + '[' + key + ']';
	                }
	                outName = Name + '[' + key + ']';
	            }
	            js_traverse(o[key], outName, key);
	        }
	        if(!isArray(o))
	            output1 = output1 + '</blockquote>}<br>';
	    }
	    else{
	        output1 = output1 + ' <input type="text" id="' + outName + '" value="' + o + '"/><br>';
	    }
	}

	function callBack(){
	    switch(req.readyState) {
	        case 4:
	            if(req.status!=200 && 0) {
	            alert("Errorjjj:"+req.status);
	            }else{
	            var output_field = document.getElementById("outputObject");
	            var output1_field = document.getElementById("output1");
	            var rdState = document.getElementById('rdState');
	            test = req.responseText;
	            output1_field.innerHTML = test;
	            try{
	                responseObject = JSON.parse(test);
	                js_traverse(responseObject,'','');
	                rdState.innerHTML = 'Ready';
	            }
	            catch (e){
	                output1 = '';
	                rdState.innerHTML = 'Error';
	            }
	            output_field.innerHTML = output1;
	            output1 = '';
	            }
	        break;

	        default:
	            return false;
	        break;
	    }
	}

	function call(){
	     //create the call

	    try{
	        req = new XMLHttpRequest();
	    }
	    catch (e){
	        try{
	            req = new ActiveXObject("Msxml2.XMLHTTP");
	        }
	        catch (e){
	            try{
	                req = new ActiveXObject("Microsoft.XMLHTTP");
	            }
	            catch (failed){
	                req = null;
	            }
	        }
	    }

	    if (req == null)
	        alert("Error creating request object!");

	    var requestString = document.getElementById('requeststring').value;
	    var readVar = document.getElementById('readVar').value;
	    var rdState = document.getElementById('rdState');
	    var ipaddress = document.getElementById('ipaddress').value;
	    //send request over GET or POST
	    if(document.getElementsByName("sendmethod")[1].checked==true){
	        var url = 'C:/xampp/xampp/htdocs/JSON/JSON-php-POST/Document.txt';
	        var url = 'http://'+ipaddress+'/read';
	        var params = readVar;
	        req.open("POST", url, true);
	        req.setRequestHeader("Content-type", "application/json");
	        req.setRequestHeader("Content-length", params.length);
	        req.setRequestHeader("Connection", "close");
	        req.onreadystatechange = callBack;
	        rdState.innerHTML = 'Reading '+readVar+' ...';
	        req.send(params);
	    }
	    else if(document.getElementsByName("sendmethod")[0].checked==true){
	        var url = 'C:/xampp/xampp/htdocs/JSON/JSON-php-POST/Document.txt';
	        var url = 'http://'+ipaddress+'/write';
	        var params = requestString;
	        req.open("POST", url, true);
	        req.setRequestHeader("Content-type", "application/json");
	        req.setRequestHeader("Content-length", params.length);
	        req.setRequestHeader("Connection", "close");
	        req.onreadystatechange = callBack;
	        rdState.innerHTML = 'Writing ...';
	        req.send(params);
	    }
	    else if(document.getElementsByName("sendmethod")[2].checked==true){
	        var url = 'C:/xampp/xampp/htdocs/JSON/JSON-php-POST/Document.txt';
	        var url = 'http://'+ipaddress+'/writetofile';
	        var params = requestString;
	        req.open("POST", url, true);
	        req.setRequestHeader("Content-type", "application/json");
	        req.setRequestHeader("Content-length", params.length);
	        req.setRequestHeader("Connection", "close");
	        req.onreadystatechange = callBack;
	        rdState.innerHTML = 'Writing to file ...';
	        req.send(params);
	    }
	}

	function pdbversion(){
	    valuesToObject(responseObject,'');
	    document.getElementById('requeststring').value = JSON.stringify(responseObject);
	}

	function pdbbrowse(){
	    document.getElementById('requeststring').value = '{ "json-rpc" : "2.0", "method" : "pdb.browse", "id" : 1}';
	}

	        </script>
	        <script type="text/javascript">

	if (!this.JSON) {
	    this.JSON = {};
	}

	(function () {

	    function f(n) {
	        // Format integers to have at least two digits.
	        return n < 10 ? '0' + n : n;
	    }

	    if (typeof Date.prototype.toJSON !== 'function') {

	        Date.prototype.toJSON = function (key) {

	            return isFinite(this.valueOf()) ?
	                   this.getUTCFullYear()   + '-' +
	                 f(this.getUTCMonth() + 1) + '-' +
	                 f(this.getUTCDate())      + 'T' +
	                 f(this.getUTCHours())     + ':' +
	                 f(this.getUTCMinutes())   + ':' +
	                 f(this.getUTCSeconds())   + 'Z' : null;
	        };

	        String.prototype.toJSON =
	        Number.prototype.toJSON =
	        Boolean.prototype.toJSON = function (key) {
	            return this.valueOf();
	        };
	    }

	    var cx = /[\u0000\u00ad\u0600-\u0604\u070f\u17b4\u17b5\u200c-\u200f\u2028-\u202f\u2060-\u206f\ufeff\ufff0-\uffff]/g,
	        escapable = /[\\\"\x00-\x1f\x7f-\x9f\u00ad\u0600-\u0604\u070f\u17b4\u17b5\u200c-\u200f\u2028-\u202f\u2060-\u206f\ufeff\ufff0-\uffff]/g,
	        gap,
	        indent,
	        meta = {    // table of character substitutions
	            '\b': '\\b',
	            '\t': '\\t',
	            '\n': '\\n',
	            '\f': '\\f',
	            '\r': '\\r',
	            '"' : '\\"',
	            '\\': '\\\\'
	        },
	        rep;

	    function quote(string) {

	        escapable.lastIndex = 0;
	        return escapable.test(string) ?
	            '"' + string.replace(escapable, function (a) {
	                var c = meta[a];
	                return typeof c === 'string' ? c :
	                    '\\u' + ('0000' + a.charCodeAt(0).toString(16)).slice(-4);
	            }) + '"' :
	            '"' + string + '"';
	    }

	    function str(key, holder) {

	        var i,          // The loop counter.
	            k,          // The member key.
	            v,          // The member value.
	            length,
	            mind = gap,
	            partial,
	            value = holder[key];

	        if (value && typeof value === 'object' &&
	                typeof value.toJSON === 'function') {
	            value = value.toJSON(key);
	        }

	        if (typeof rep === 'function') {
	            value = rep.call(holder, key, value);
	        }

	        switch (typeof value) {
	        case 'string':
	            return quote(value);

	        case 'number':

	            return isFinite(value) ? String(value) : 'null';

	        case 'boolean':
	        case 'null':

	            return String(value);

	        case 'object':

	            if (!value) {
	                return 'null';
	            }

	            gap += indent;
	            partial = [];

	            if (Object.prototype.toString.apply(value) === '[object Array]') {

	                length = value.length;
	                for (i = 0; i < length; i += 1) {
	                    partial[i] = str(i, value) || 'null';
	                }

	                v = partial.length === 0 ? '[]' :
	                    gap ? '[\n' + gap +
	                            partial.join(',\n' + gap) + '\n' +
	                                mind + ']' :
	                          '[' + partial.join(',') + ']';
	                gap = mind;
	                return v;
	            }

	            if (rep && typeof rep === 'object') {
	                length = rep.length;
	                for (i = 0; i < length; i += 1) {
	                    k = rep[i];
	                    if (typeof k === 'string') {
	                        v = str(k, value);
	                        if (v) {
	                            partial.push(quote(k) + (gap ? ': ' : ':') + v);
	                        }
	                    }
	                }
	            } else {

	                for (k in value) {
	                    if (Object.hasOwnProperty.call(value, k)) {
	                        v = str(k, value);
	                        if (v) {
	                            partial.push(quote(k) + (gap ? ': ' : ':') + v);
	                        }
	                    }
	                }
	            }

	            v = partial.length === 0 ? '{}' :
	                gap ? '{\n' + gap + partial.join(',\n' + gap) + '\n' +
	                        mind + '}' : '{' + partial.join(',') + '}';
	            gap = mind;
	            return v;
	        }
	    }

	    if (typeof JSON.stringify !== 'function') {
	        JSON.stringify = function (value, replacer, space) {

	            var i;
	            gap = '';
	            indent = '';

	            if (typeof space === 'number') {
	                for (i = 0; i < space; i += 1) {
	                    indent += ' ';
	                }

	            } else if (typeof space === 'string') {
	                indent = space;
	            }

	            rep = replacer;
	            if (replacer && typeof replacer !== 'function' &&
	                    (typeof replacer !== 'object' ||
	                     typeof replacer.length !== 'number')) {
	                throw new Error('JSON.stringify');
	            }

	            return str('', {'': value});
	        };
	    }

	    if (typeof JSON.parse !== 'function') {
	        JSON.parse = function (text, reviver) {

	            var j;

	            function walk(holder, key) {

	                var k, v, value = holder[key];
	                if (value && typeof value === 'object') {
	                    for (k in value) {
	                        if (Object.hasOwnProperty.call(value, k)) {
	                            v = walk(value, k);
	                            if (v !== undefined) {
	                                value[k] = v;
	                            } else {
	                                delete value[k];
	                            }
	                        }
	                    }
	                }
	                return reviver.call(holder, key, value);
	            }

	            text = String(text);
	            cx.lastIndex = 0;
	            if (cx.test(text)) {
	                text = text.replace(cx, function (a) {
	                    return '\\u' +
	                        ('0000' + a.charCodeAt(0).toString(16)).slice(-4);
	                });
	            }

	            if (/^[\],:{}\s]*$/
	.test(text.replace(/\\(?:["\\\/bfnrt]|u[0-9a-fA-F]{4})/g, '@')
	.replace(/"[^"\\\n\r]*"|true|false|null|-?\d+(?:\.\d*)?(?:[eE][+\-]?\d+)?/g, ']')
	.replace(/(?:^|:|,)(?:\s*\[)+/g, ''))) {

	                j = eval('(' + text + ')');

	                return typeof reviver === 'function' ?
	                    walk({'': j}, '') : j;
	            }

	            throw new SyntaxError('JSON.parse');
	        };
	    }
	}());

	        </script>

	    </head>
	<body>
	<div style="text-align:center;">
	<table style="width: 800px; margin-left: auto;
	margin-right: auto;" border="0" cellpadding="0" cellspacing="0">
	  <tbody>
	    <tr>
	      <td style="height: 50px; background-color: rgb(255, 131, 0);"><font size="+2">&nbsp;<span style="font-weight: bold; font-size : 20pt;">BRSE JSON</span></font></td>
	    </tr>
	    <tr>
	      <td style="height: 10px; background-color: rgb(102, 102, 102);"></td>
	    </tr>
	    <tr>
	      <td>
	      <table style="width: 100%; border-collapse: collapse;" border="1" bordercolor="#666666" cellpadding="5" cellspacing="0"><tr><td style="background-color: rgb(204, 204, 204);">
		        Outgoing JSON: <br>
	            <textarea cols="95" rows="10" id="requeststring"></textarea><br />
		        Variable to Read: <input type="text" id="readVar" value="PV_var1"/><br />
		        IP Address: <input type="text" id="ipaddress" value="10.46.10.211"/><br />
	            Method: <input type="radio" name="sendmethod" value="POST"> WRITE
	                <input type="radio" name="sendmethod" value="POST" checked> READ
	                <input type="radio" name="sendmethod" value="POST"> WRITE TO FILE<br>
	                <input type="submit" value="Send" onclick="call();" />
	                <input type="submit" value="Build Output" onclick="pdbversion();" /><br>
	            <br />
	            Status: <b id="rdState" style="color:black"></b><br>
	            </td>
	            </tr>
	            <tr><td>
	            <div id="outputObject"></div><br>
	            <div id="output1" style="color:green; word-break:break-all; word-wrap:break-word;"></div>
	            </td>
	            </tr>
	            <tr>
	            <td>
	            </td>
	            </tr>
	      </table>
	      </td>
	    </tr>
	    <tr>
	      <td style="height: 5px; background-color: rgb(102, 102, 102);"></td>
	    </tr>
	  </tbody>
	</table>
	</div>

	    </body>
	</html>
\endcode

*/
```

#### version_history.c
```c
/*!\file version_history.c */

/*!
	\page History
	\section History

	\par V1.00.0
		\arg March 2011 Created by Damerow

	\par V1.00.1
		\arg 14 April 2011 Helpfile and example added. First release version. (Valdt)

    \par V1.1  (Yueming)
		\arg Library dependency changed from AsString to AsBrStr.
             Add #include <AsBrStr.h>
        \arg Functions atof, ftoa, atoi and itoa are changed to brsatof, brsftoa, brsatoi, and brsitoa
             to avoid name conflict.
        \arg Functions strcat and strcpy can continue to be used from string.h

*/
```

### Library Logical/Libraries/Queue (IEC)

#### Types.typ - Exported data types
```iecst
TYPE
	FifoQueue_typ : 	STRUCT
		NextAvailableIndex : UDINT;
		Queue : ARRAY[0..QUEUE_SIZE_M1]OF Data_typ;
	END_STRUCT;
	Data_typ : 	STRUCT
		Data : ARRAY[0..MAX_DATA_LENGTH_M1]OF USINT;
	END_STRUCT;
	FifoLogQueue_typ : 	STRUCT
		NextAvailableIndex : UDINT;
		Queue : ARRAY[0..QUEUE_SIZE_M1]OF Data_Log_typ;
	END_STRUCT;
	Data_Log_typ : 	STRUCT
		Data : ARRAY[0..MAX_DATA_LOG_LENGTH_M1]OF USINT;
	END_STRUCT;
END_TYPE
```

#### Constants.var - Exported constants
```iecst
VAR CONSTANT
	QUEUE_SIZE : UDINT := 200;
	QUEUE_SIZE_M1 : UDINT := QUEUE_SIZE - 1;
	MAX_DATA_LENGTH_M1 : UINT := MAX_DATA_LENGTH-1;
	MAX_DATA_LENGTH : UINT := 1000;
	MAX_DATA_LOG_LENGTH : UINT := 10080;
	MAX_DATA_LOG_LENGTH_M1 : UINT := MAX_DATA_LOG_LENGTH-1;
END_VAR
```

#### Queue.fun - Exported functions and function blocks
```iecst
{REDUND_ERROR} FUNCTION FifoPush : BOOL (*TODO: Add your comment here*) (*$GROUP=User,$CAT=User,$GROUPICON=User.png,$CATICON=User.png*)
	VAR_INPUT
		Queue : REFERENCE TO FifoQueue_typ;
		Value : Data_typ;
	END_VAR
END_FUNCTION

{REDUND_ERROR} FUNCTION FifoPop : UINT (*TODO: Add your comment here*) (*$GROUP=User,$CAT=User,$GROUPICON=User.png,$CATICON=User.png*)
	VAR_INPUT
		Queue : REFERENCE TO FifoQueue_typ;
	END_VAR
END_FUNCTION

{REDUND_ERROR} FUNCTION FifoReset : BOOL (*TODO: Add your comment here*) (*$GROUP=User,$CAT=User,$GROUPICON=User.png,$CATICON=User.png*)
	VAR_INPUT
		Queue : REFERENCE TO FifoQueue_typ;
	END_VAR
END_FUNCTION

{REDUND_ERROR} FUNCTION FifoPushLog : BOOL (*TODO: Add your comment here*) (*$GROUP=User,$CAT=User,$GROUPICON=User.png,$CATICON=User.png*)
	VAR_INPUT
		Queue : REFERENCE TO FifoLogQueue_typ;
		Value : Data_Log_typ;
	END_VAR
END_FUNCTION

{REDUND_ERROR} FUNCTION FifoPopLog : UINT (*TODO: Add your comment here*) (*$GROUP=User,$CAT=User,$GROUPICON=User.png,$CATICON=User.png*)
	VAR_INPUT
		Queue : REFERENCE TO FifoLogQueue_typ;
	END_VAR
END_FUNCTION

{REDUND_ERROR} FUNCTION FifoResetLog : BOOL (*TODO: Add your comment here*) (*$GROUP=User,$CAT=User,$GROUPICON=User.png,$CATICON=User.png*)
	VAR_INPUT
		Queue : REFERENCE TO FifoLogQueue_typ;
	END_VAR
END_FUNCTION
```

#### FifoPush.st
```iecst
(* TODO: Add your comment here *)
FUNCTION FifoPush

	Queue.Queue[Queue.NextAvailableIndex] := Value;

	Queue.NextAvailableIndex := Queue.NextAvailableIndex + 1;

	IF Queue.NextAvailableIndex > QUEUE_SIZE_M1 THEN
		Queue.NextAvailableIndex := QUEUE_SIZE_M1;
	END_IF

	FifoPush := TRUE;

END_FUNCTION
```

#### FifoPop.st
```iecst
(* TODO: Add your comment here *)
FUNCTION FifoPop

	//we want to return something more complex than a basic data type but we can't. Instead, just use pop to remove the top item without returning it
	FifoPop := 0;
	//FifoPop := Queue.Queue[0];

	brsmemmove(ADR(Queue.Queue[0]), ADR(Queue.Queue[1]), SIZEOF(Queue.Queue) - SIZEOF(Queue.Queue[0]));

	IF Queue.NextAvailableIndex > 0 THEN
		Queue.NextAvailableIndex := Queue.NextAvailableIndex - 1;
	END_IF

END_FUNCTION
```

#### FifoReset.st
```iecst
(* TODO: Add your comment here *)
FUNCTION FifoReset

	brsmemset(ADR(Queue), 0, SIZEOF(Queue));

	FifoReset := TRUE;

END_FUNCTION
```

#### FifoPushLog.st
```iecst
(* TODO: Add your comment here *)
FUNCTION FifoPushLog

	Queue.Queue[Queue.NextAvailableIndex] := Value;

	Queue.NextAvailableIndex := Queue.NextAvailableIndex + 1;

	IF Queue.NextAvailableIndex > QUEUE_SIZE_M1 THEN
		Queue.NextAvailableIndex := QUEUE_SIZE_M1;
	END_IF

	FifoPushLog := TRUE;

END_FUNCTION
```

#### FifoPopLog.st
```iecst
(* TODO: Add your comment here *)
FUNCTION FifoPopLog

	//we want to return something more complex than a basic data type but we can't. Instead, just use pop to remove the top item without returning it
	FifoPopLog := 0;
	//FifoPop := Queue.Queue[0];

	brsmemmove(ADR(Queue.Queue[0]), ADR(Queue.Queue[1]), SIZEOF(Queue.Queue) - SIZEOF(Queue.Queue[0]));

	IF Queue.NextAvailableIndex > 0 THEN
		Queue.NextAvailableIndex := Queue.NextAvailableIndex - 1;
	END_IF

END_FUNCTION
```

#### FifoResetLog.st
```iecst
(* TODO: Add your comment here *)
FUNCTION FifoResetLog

	brsmemset(ADR(Queue), 0, SIZEOF(Queue));

	FifoResetLog := TRUE;

END_FUNCTION
```

### LibAsTCP1_ST.typ
```iecst
(********************************************************************
 * COPYRIGHT -- Bernecker + Rainer
 ********************************************************************
 * Package: LibAsTCP
 * File: LibAsTCP.typ
 * Author: Bernecker + Rainer
 * Created: February 21, 2008
 ********************************************************************
 * Data types of package LibAsTCP
 ********************************************************************)

TYPE
	LibAsTCP1_ST_typ : 	STRUCT  (*Datatyp for global Variables*)
		receive_data : ARRAY[0..400]OF USINT; (*Data which has been received*)
		send_data : ARRAY[0..100]OF UDINT; (*Data which should be sent*)
	END_STRUCT;
END_TYPE
```

### Program Logical/TCPComms/Client

#### Client.var
```iecst
(********************************************************************
 * COPYRIGHT -- Bernecker + Rainer
 ********************************************************************
 * Package: LibAsTCP
 * File: LibAsTCP.var
 * Author: Bernecker + Rainer
 * Created: February 21, 2008
 ********************************************************************
 * Variables of package LibAsTCP
 ********************************************************************)
VAR
	ReconnectWait : BOOL;
	ClientConnected : BOOL;
	TON_Reopen : TON;
	Client : Client_typ := (0); (*Data for Client Task*)
	ServerPort : UINT;
	ServerIP : STRING[20];
	SendData : Data_typ;
	prevStep : UINT;
	message_tmp : Data_typ;
	CreateTestMessage1 : BOOL;
	JSON_Stringify_0 : JSON_Stringify;
END_VAR
```

#### Client.st
```iecst
(********************************************************************
 * COPYRIGHT -- Bernecker + Rainer
 ********************************************************************
 * Program: Client
 * File: Client.st
 * Author: Bernecker + Rainer
 * Created: February 21, 2008
 ********************************************************************
 * Implementation of program Client
 ********************************************************************)
PROGRAM _INIT

	//blank out queue just in case it initializes with non-zero info
	FifoReset(ADR(gSendQueue));
	TON_Reopen.PT := t#10s;

	ServerIP := '127.0.0.1';
	//ServerIP := '192.168.0.102';
	ServerPort := 9999;

	gMessageToEZ3.Move_Command := 'Auto_Run';
	gMessageToEZ3.Battery_Subscribe := 1;

END_PROGRAM

PROGRAM _CYCLIC

	IF CreateTestMessage1 THEN
		CreateTestMessage1 := FALSE;

		//brsmemset(ADR(gMessageToEZ3), 0, SIZEOF(gMessageToEZ3));

		brsmemset(ADR(message_tmp), 0, SIZEOF(message_tmp));
		brsmemset(ADR(JSON_Stringify_0),0,SIZEOF(JSON_Stringify_0));;

		REPEAT
			JSON_Stringify_0(pStName := ADR('gMessageToEZ3'));
			brsstrcat(ADR(message_tmp),ADR(JSON_Stringify_0.Output));
			UNTIL JSON_Stringify_0.Status <> 0
		END_REPEAT;

		FifoPush(ADR(gSendQueue), message_tmp);
	END_IF

	CASE Client.sStep OF

		0: (* Open Ethernet Interface *)
			prevStep := Client.sStep;
			Client.TcpOpen_0.enable := 1;
			Client.TcpOpen_0.pIfAddr := 0;  (* Which Interface to open *)
			Client.TcpOpen_0.port := 12001;  (* Port on client side to use *)
			Client.TcpOpen_0.options := 0;
			Client.TcpOpen_0;  (* Call the Function *)

			IF Client.TcpOpen_0.status = 0 THEN  (* TcpOpen successfull *)
				Client.sStep := 5;
			ELSIF Client.TcpOpen_0.status = ERR_FUB_BUSY THEN  (* TcpOpen not finished -> redo *)
				(* Busy *)
			ELSE  (* Goto Error Step *)
				prevStep := Client.sStep;
				Client.sStep := 100;
			END_IF

		5:
			prevStep := Client.sStep;
			Client.linger_opt.lLinger := 0; (* linger Time = 0 *)
			Client.linger_opt.lOnOff := 0; (* linger Option OFF *)

			Client.TcpIoctl_0.enable := 1;
			Client.TcpIoctl_0.ident := Client.TcpOpen_0.ident; (* Connection Ident from AsTP.TCP_Open *)
			Client.TcpIoctl_0.ioctl := tcpSO_LINGER_SET; (* Set Linger Options *)
			Client.TcpIoctl_0.pData := ADR(Client.linger_opt);
			Client.TcpIoctl_0.datalen := SIZEOF(Client.linger_opt);
			Client.TcpIoctl_0;

			IF Client.TcpIoctl_0.status = 0 THEN  (* TcpIoctl successfull *)
				Client.sStep := 10;
			ELSIF Client.TcpIoctl_0.status = ERR_FUB_BUSY THEN  (* TcpIoctl not finished -> redo *)
				(* Busy *)
			ELSE  (* Goto Error Step *)
				Client.sStep := 100;
			END_IF

		10: (* Connect to the other Station *)
			prevStep := Client.sStep;
			Client.TcpClient_0.enable := 1;
			Client.TcpClient_0.ident := Client.TcpOpen_0.ident;  (* Connection Ident from AsTCP.TCP_Open *)
			Client.TcpClient_0.portserv := ServerPort;  (* Port on server side to use *)
			Client.TcpClient_0.pServer := ADR(ServerIP);  (* Server Address *)
			Client.TcpClient_0;  (* Call the Function*)

			IF Client.TcpClient_0.status = 0 THEN  (* Open ok -> Send Data *)
				Client.sStep := 15;
			ELSIF Client.TcpClient_0.status = ERR_FUB_BUSY THEN  (* TcpClient not finished -> redo *)
				(* Busy *)
			ELSIF Client.TcpClient_0.status = tcpERR_INVALID THEN  (* Port error -> Close actual connection, and reopen a new one in 10s *)
				Client.sStep := 40;
				ReconnectWait := TRUE;
			ELSE  (* Goto Error Step *)
				Client.sStep := 100;
			END_IF

		15:
			IF gSendQueue.NextAvailableIndex > 0 THEN
				// copy the top item of the queue and then pop it
				// our functions can't return non-basic types, so I can't pop right into the send data - JDL
				brsmemset(ADR(SendData), 0, SIZEOF(SendData));
				brsmemcpy(ADR(SendData), ADR(gSendQueue.Queue[0]), SIZEOF(SendData));

				Client.sStep := 20;
			END_IF

		20: (* Send Data to the Server *)
			prevStep := Client.sStep;

			Client.TcpSend_0.enable := 1;
			Client.TcpSend_0.ident := Client.TcpOpen_0.ident;  (* Connection Ident from AsTCP.TCP_Open *)
			Client.TcpSend_0.pData := ADR(SendData);  (* Which data to send *)
			Client.TcpSend_0.datalen := brsstrlen(ADR(SendData));  (* Lenght of data to send *)
			Client.TcpSend_0.flags := 0;
			Client.TcpSend_0;  (* Call the Function*)

			IF Client.TcpSend_0.status = 0 THEN  (* Data was sent sucessfully -> receive data *)
				FifoPop(ADR(gSendQueue));
				Client.sStep := 30;
			ELSIF Client.TcpSend_0.status = ERR_FUB_BUSY THEN  (* TcpSend not finished -> redo *)
				(* Busy *)
			ELSIF (Client.TcpSend_0.status = tcpERR_SENTLEN) OR (Client.TcpSend_0.status = tcpERR_NOT_CONNECTED) THEN (* Connection Lost *)
				Client.sStep := 40;
			ELSE  (* Goto Error Step *)
				Client.sStep := 100;
			END_IF

		30: (* Receive Data from the Server *)
			prevStep := Client.sStep;
			Client.TcpRecv_0.enable := 1;
			Client.TcpRecv_0.ident := Client.TcpOpen_0.ident;  (* Connection Ident from AsTCP.TCP_Open *)
			Client.TcpRecv_0.pData	:= ADR(LibAsTCP1_ST.receive_data);  (* Where to store the incoming data *)
			Client.TcpRecv_0.datamax := SIZEOF(LibAsTCP1_ST.receive_data);  (* Lenght of data buffer *)
			Client.TcpRecv_0.flags := 0;
			Client.TcpRecv_0;  (* Call the Function*)

			IF Client.TcpRecv_0.status = 0 THEN  (* Data was received sucessfully -> Send next packet *)
				Client.sStep := 15;
				Client.recv_timeout := 0;
			ELSIF Client.TcpRecv_0.status = 0 THEN  (* Data was received sucessfully, but Message number not matched. Resend packet *)
				Client.sStep := 15;
				Client.recv_timeout := 0;
			ELSIF Client.TcpRecv_0.status = tcpERR_NO_DATA THEN  (* No data received - wait *)
				Client.recv_timeout := Client.recv_timeout + 1;
				IF Client.recv_timeout > 100 THEN //5s
				//	Client.sStep := 40;
					Client.sStep := 15;
					ReconnectWait := TRUE;
					Client.recv_timeout := 0;
				END_IF
				(* No Data received *)
			ELSIF Client.TcpRecv_0.status = ERR_FUB_BUSY THEN  (* TcpRecv not finished -> redo *)
				(* Busy *)
			ELSIF Client.TcpRecv_0.status = tcpERR_NOT_CONNECTED THEN (* Connection Lost *)
				Client.sStep := 40;
			ELSE  (* Goto Error Step *)
				Client.sStep := 100;
			END_IF

		40: (* Close connection *)
			prevStep := Client.sStep;
			Client.TcpClose_0.enable := 1;
			Client.TcpClose_0.ident := Client.TcpOpen_0.ident;  (* Connection Ident from AsTCP.TCP_Open *)
			Client.TcpClose_0.how := 0;
			Client.TcpClose_0;  (* Call the Function*)

			IF Client.TcpClose_0.status = 0 AND NOT ReconnectWait THEN  (* Close sucessfull -> Reopen the interface *)
				Client.sStep := 0;
			ELSIF Client.TcpClose_0.status = 0 AND ReconnectWait THEN  (* Close sucessfull -> Reopen the interface w/ 10s delay *)
				Client.sStep := 50;
				ReconnectWait := FALSE;
			ELSIF Client.TcpClose_0.status = ERR_FUB_BUSY THEN  (* TcpClose not finished -> redo *)
				(* Busy *)
			ELSE  (* Goto Error Step *)
				Client.sStep := 100;
			END_IF

		50: (*Wait to reopen connection*)
			TON_Reopen.IN := TRUE;
			IF TON_Reopen.Q THEN
				Client.sStep := 0;
				TON_Reopen.IN := FALSE;
			END_IF

		100: (* Error State. Wait 10s, try again *)
			TON_Reopen.IN := TRUE;
			IF TON_Reopen.Q THEN
				Client.sStep := prevStep;
				TON_Reopen.IN := FALSE;
			END_IF

	END_CASE

	TON_Reopen();

END_PROGRAM
```

### Program Logical/TCPComms/Server

#### Server.var
```iecst
(********************************************************************
 * COPYRIGHT -- Bernecker + Rainer
 ********************************************************************
 * Package: LibAsTCP
 * File: LibAsTCP.var
 * Author: Bernecker + Rainer
 * Created: February 21, 2008
 ********************************************************************
 * Variables of package LibAsTCP
 ********************************************************************)
VAR
	Data : Data_typ;
	ShuttleRoute : ARRAY[0..20] OF USINT;
	TempSeqNum : UDINT;
	j : USINT;
	i : USINT;
	RouteBoolArray : ARRAY[0..63] OF BOOL;
	TON_MessageTimeout : TON;
	OwnPort : UINT;
	Server : Server_typ := (0); (*Data for Server Task*)
	VariablesNotFound : ARRAY[0..29] OF STRING[50];
	Debug : ARRAY[0..29] OF STRING[50];
	MessageData : Data_typ;
	MessageSize : UDINT;
	MessageType : UDINT;
	RouteUINTArray : ARRAY[0..63] OF UINT;
	Byte2Bit_0 : Byte2Bit;
	prevStep : UINT;
	TON_Reopen : TON;
	LogQueueData : Data_typ;
	LogMessageData : EventLog_Event_typ;
	shuttleID_int : UINT;
	shuttleLoc_int : UDINT;
	shuttleLoc : STRING[4];
	shuttleID : STRING[4];
	routeStep : STRING[4];
END_VAR
```

#### Server.st
```iecst
(********************************************************************
 * COPYRIGHT -- Bernecker + Rainer
 ********************************************************************
 * Program: Server
 * File: Server.st
 * Author: Bernecker + Rainer
 * Created: February 21, 2008
 ********************************************************************
 * Implementation of program Server
 ********************************************************************)
PROGRAM _INIT

	OwnPort := 3000;
	//OwnPort := 10000;
	Server.client_address := '127.0.0.1';
	TON_Reopen.PT := t#10s;
	TON_MessageTimeout.PT := t#100ms;

END_PROGRAM

PROGRAM _CYCLIC

	//Server Idle Status
	gServerIdle := Server.sStep = 20;

	CASE Server.sStep OF

		0:  (* Open Ethernet Interface *)
			prevStep := Server.sStep;
			Server.TcpOpen_0.enable := 1;
			Server.TcpOpen_0.pIfAddr := 0;  (* Listen on all TCP/IP Interfaces*)
			Server.TcpOpen_0.port := OwnPort;  (* Port to listen*)
			Server.TcpOpen_0.options := 0;
			Server.TcpOpen_0;  (* Call the Function*)

			IF Server.TcpOpen_0.status = 0 THEN  (* TcpOpen successfull*)
				Server.sStep := 5;
			ELSIF Server.TcpOpen_0.status = ERR_FUB_BUSY THEN  (* TcpOpen not finished -> redo *)
			  (* Busy *)
			ELSE  (* Goto Error Step *)
				Server.sStep := 100;
			END_IF

		5:
			prevStep := Server.sStep;
			Server.linger_opt.lLinger := 0; (* linger Time = 0 *)
			Server.linger_opt.lOnOff := 0; (* linger Option OFF *)

		 	Server.TcpIoctl_0.enable := 1;
			Server.TcpIoctl_0.ident := Server.TcpOpen_0.ident; (* Connection Ident from AsTCP.TCP_Open *)
			Server.TcpIoctl_0.ioctl := tcpSO_LINGER_SET; (* Set Linger Options *)
			Server.TcpIoctl_0.pData := ADR(Server.linger_opt);
			Server.TcpIoctl_0.datalen := SIZEOF(Server.linger_opt);
   			Server.TcpIoctl_0;

			IF Server.TcpIoctl_0.status = 0 THEN  (* TcpIoctl successfull *)
				Server.sStep := 10;
			ELSIF Server.TcpIoctl_0.status = ERR_FUB_BUSY THEN  (* TcpIoctl not finished -> redo *)
			  (* Busy *)
			ELSE  (* Goto Error Step *)
				Server.sStep := 100;
			END_IF

		10: (* Wait for Client Connection *)
			prevStep := Server.sStep;
			Server.TcpServer_0.enable := 1;
			Server.TcpServer_0.ident := Server.TcpOpen_0.ident;  (* Connection Ident from AsTCP.TCP_Open *)
			Server.TcpServer_0.backlog := 1;  (* Number of clients waiting simultaneously for a connection*)
			Server.TcpServer_0.pIpAddr := ADR(Server.client_address);  (* Where to write the client IP-Address*)
			Server.TcpServer_0;  (* Call the Function*)

			IF Server.TcpServer_0.status = 0 THEN  (* Status = 0 if an client connects to server *)
				Server.sStep := 15;
			ELSIF Server.TcpServer_0.status = ERR_FUB_BUSY THEN  (* TcpServer not finished -> redo *)
			  (* Busy *)
			ELSE  (* Goto Error Step *)
				Server.sStep := 100;
			END_IF

		15:
			prevStep := Server.sStep;
		 	Server.TcpIoctl_0.enable := 1;
			Server.TcpIoctl_0.ident := Server.TcpServer_0.identclnt; (* Connection Ident from AsTCP.TCP_Server *)
			Server.TcpIoctl_0.ioctl := tcpSO_LINGER_SET;  (* Set Linger Options *)
			Server.TcpIoctl_0.pData := ADR(Server.linger_opt);
			Server.TcpIoctl_0.datalen := SIZEOF(Server.linger_opt);
   			Server.TcpIoctl_0;

			IF Server.TcpIoctl_0.status = 0 THEN  (* TcpIoctl successfull *)
				Server.sStep := 20;
			ELSIF Server.TcpIoctl_0.status = ERR_FUB_BUSY THEN  (* TcpIoctl not finished -> redo *)
			  (* Busy *)
			ELSE  (* Goto Error Step *)
				Server.sStep := 100;
			END_IF

		20: (* Wait for Data *)
			prevStep := Server.sStep;
			Server.TcpRecv_0.enable := 1;
			Server.TcpRecv_0.ident := Server.TcpServer_0.identclnt;  (* Client Ident from AsTCP.TCP_Server *)
			Server.TcpRecv_0.pData	:= ADR(Server.data_buffer);  (* Where to store the incoming data *)
			Server.TcpRecv_0.datamax := SIZEOF(Server.data_buffer);  (* Lenght of data buffer *)
			Server.TcpRecv_0.flags := 0;
			Server.TcpRecv_0;  (* Call the Function*)

			IF Server.TcpRecv_0.status = 0 AND (Server.data_buffer[1] = 0 OR Server.data_buffer[1] = (gMessageSequenceNumberServer)) THEN  (* Data received and Message count match*)

				Server.recv_timeout := 0;

				//Log Received message based on type
				brsmemset(ADR(LogMessageData.AdditionalData), 0, SIZEOF(LogMessageData.AdditionalData));
				brsmemset(ADR(LogQueueData), 0, SIZEOF(LogQueueData));
				LogMessageData.AdditionalDataFormat := arEVENTLOG_ADDFORMAT_TEXT;
				LogMessageData.EnteredBy := 'B&R Msg In';
				LogMessageData.EventID := ArEventLogMakeEventID(Severity := arEVENTLOG_SEVERITY_INFO, Facility := UDINT_TO_UINT(Server.data_buffer[2]), ErrorCode := 0);

				CASE Server.data_buffer[2] OF

					0: //Heartbeat
						LogMessageData.AdditionalData := 'Heartbeat';
						Server.sStep := 30;

					1: //Reset after error
						gProcess.Commands.Reset := TRUE;
						LogMessageData.AdditionalData := 'Error Reset';
						Server.sStep := 30;

					2: //Start the Track
						gProcess.Commands.PowerOn := TRUE;
						LogMessageData.AdditionalData := 'Trak Power On';
						Server.sStep := 30;

					3: //Run the Track
						gProcess.Commands.Start := TRUE;
						LogMessageData.AdditionalData := 'Trak Start';
						Server.sStep := 30;

					4: //Stop the Track
						gProcess.Commands.Stop := TRUE;
						LogMessageData.AdditionalData := 'Trak Stop';
						gProcess.Status.StoppedTrack := Server.data_buffer[4];
						Server.sStep := 30;

					5: //Request shuttle to a Carton insert station.
						brsmemcpy(ADR(RouteUINTArray),ADR(Server.data_buffer[4]), 8);
						Byte2Bit_0(byteadr := ADR(RouteUINTArray[0]), length := 16); (* convert byte array into bit array *)
						brsmemcpy(ADR(RouteBoolArray[0]), Byte2Bit_0.bitadr, 16);
						Byte2Bit_0(byteadr := ADR(RouteUINTArray[1]), length := 16); (* convert byte array into bit array *)
						brsmemcpy(ADR(RouteBoolArray[16]), Byte2Bit_0.bitadr, 16);
						Byte2Bit_0(byteadr := ADR(RouteUINTArray[2]), length := 16); (* convert byte array into bit array *)
						brsmemcpy(ADR(RouteBoolArray[32]), Byte2Bit_0.bitadr, 16);
						Byte2Bit_0(byteadr := ADR(RouteUINTArray[3]), length := 16); (* convert byte array into bit array *)
						brsmemcpy(ADR(RouteBoolArray[48]), Byte2Bit_0.bitadr, 16);

						LogMessageData.AdditionalData := 'Shuttle Request, Shuttle Route: ';

						j := 0;
						FOR i := 0 TO 63 DO
							IF RouteBoolArray[i] = TRUE THEN
								ShuttleRoute[j] := i;
								j := j + 1;
								routeStep := INT_TO_STRING(i);
								brsstrcat(ADR(LogMessageData.AdditionalData), ADR(routeStep));
								brsstrcat(ADR(LogMessageData.AdditionalData), ADR(' '));
							END_IF
						END_FOR;
						ShuttleRoute[j] := UDINT_TO_USINT(SCAN);
						brsmemcpy(ADR(Data),ADR(ShuttleRoute),SIZEOF(ShuttleRoute));
						FifoPush(ADR(gShutReqQueue), Data);
						Server.sStep := 30;

					7: //Release shuttle from station
						IF (gShuttleIDAtLocation[Server.data_buffer[5]] <> 0) THEN
							gReleaseFromStation[Server.data_buffer[5]] := TRUE;
						END_IF

						LogMessageData.AdditionalData := 'Release Shuttle, ';
						brsstrcat(ADR(LogMessageData.AdditionalData), ADR('Shuttle ID: '));
						brsmemcpy(ADR(shuttleID_int), ADR(gShuttleIDAtLocation[Server.data_buffer[5]]), 4);
						shuttleID := INT_TO_STRING(shuttleID_int);
						brsstrcat(ADR(LogMessageData.AdditionalData), ADR(shuttleID));
						brsstrcat(ADR(LogMessageData.AdditionalData), ADR(' Shuttle Loc: '));
						brsmemcpy(ADR(shuttleLoc_int), ADR(Server.data_buffer[5]), 8);
						shuttleLoc := UDINT_TO_STRING(shuttleLoc_int);
						brsstrcat(ADR(LogMessageData.AdditionalData), ADR(shuttleLoc));

						Server.sStep := 30;

					9: //Shuttle Route

						//brsmemcpy(ADR(gShuttleRoutes[Server.data_buffer[4], 0]), ADR(Server.data_buffer[5]), 8);
						brsmemcpy(ADR(RouteUINTArray),ADR(Server.data_buffer[5]), 8);
						Byte2Bit_0(byteadr := ADR(RouteUINTArray[0]), length := 16); (* convert byte array into bit array *)
						brsmemcpy(ADR(RouteBoolArray[0]), Byte2Bit_0.bitadr, 16);
						Byte2Bit_0(byteadr := ADR(RouteUINTArray[1]), length := 16); (* convert byte array into bit array *)
						brsmemcpy(ADR(RouteBoolArray[16]), Byte2Bit_0.bitadr, 16);
						Byte2Bit_0(byteadr := ADR(RouteUINTArray[2]), length := 16); (* convert byte array into bit array *)
						brsmemcpy(ADR(RouteBoolArray[32]), Byte2Bit_0.bitadr, 16);
						Byte2Bit_0(byteadr := ADR(RouteUINTArray[3]), length := 16); (* convert byte array into bit array *)
						brsmemcpy(ADR(RouteBoolArray[48]), Byte2Bit_0.bitadr, 16);

						LogMessageData.AdditionalData := 'Route Decision, Shuttle Route: ';

						j := 0;
						FOR i := 0 TO 63 DO
							IF RouteBoolArray[i] = TRUE THEN
								gShuttleRoutes[Server.data_buffer[4], j] := i;
								j := j + 1;
								routeStep := INT_TO_STRING(i);
								brsstrcat(ADR(LogMessageData.AdditionalData), ADR(routeStep));
								brsstrcat(ADR(LogMessageData.AdditionalData), ADR(' '));
							END_IF
						END_FOR;

						brsstrcat(ADR(LogMessageData.AdditionalData), ADR(' ShuttleID: '));
						brsmemcpy(ADR(shuttleID_int), ADR(Server.data_buffer[4]), 4);
						shuttleID := INT_TO_STRING(shuttleID_int);
						brsstrcat(ADR(LogMessageData.AdditionalData), ADR(shuttleID));

						gRouteRecieved[Server.data_buffer[4]] := TRUE;
						gBypassLHD[Server.data_buffer[4]] := FALSE;
						Server.sStep := 30;

					11: //Bypass Lid Hold Down

						LogMessageData.AdditionalData := 'Bypass Lid Hold-down, Shuttle ID: ';
						brsmemcpy(ADR(shuttleID_int), ADR(Server.data_buffer[4]), 4);
						shuttleID := INT_TO_STRING(shuttleID_int);
						brsstrcat(ADR(LogMessageData.AdditionalData), ADR(shuttleID));

						gBypassLHD[Server.data_buffer[4]] := TRUE;
						Server.sStep := 30;

					ELSE
						//Add error message (TODO)
						Server.sStep := 30;

				END_CASE

				//Log message if it is not heartbeat
				IF Server.data_buffer[2] <> 0 THEN
					LogMessageData.AdditionalDataSize := LEN(LogMessageData.AdditionalData);
					brsmemcpy(ADR(LogQueueData), ADR(LogMessageData), SIZEOF(LogMessageData));
					FifoPush(ADR(gLogQueue), LogQueueData);
				END_IF

				//Add ACK message
				brsmemset(ADR(Server.data_buffer), 0, SIZEOF(Server.data_buffer));
				Server.data_buffer[0] := 0;
				Server.data_buffer[1] := gMessageSequenceNumberServer;

				gMessageSequenceNumberServer := Server.data_buffer[1] + 1;

			ELSIF Server.TcpRecv_0.status = 0 AND (Server.data_buffer[1] = (gMessageSequenceNumberServer - 1)) THEN  (* Data received and Message count is previous sequence number *)
				//Send ACK
				brsmemset(ADR(Server.data_buffer), 0, SIZEOF(Server.data_buffer));
				Server.data_buffer[0] := 0;
				Server.data_buffer[1] := gMessageSequenceNumberServer - 1;
				gMessageSequenceNumberServer := Server.data_buffer[1] + 1;
				Server.sStep := 30;

			ELSIF Server.TcpRecv_0.status = 0 AND NOT(Server.data_buffer[1] = 0 OR Server.data_buffer[1] = (gMessageSequenceNumberServer)) THEN  (* Data received and Message count mismatch*)
				//Add NAK message. Will need to implement specific error codes
				TempSeqNum := Server.data_buffer[1];
				brsmemset(ADR(Server.data_buffer), 0, SIZEOF(Server.data_buffer));
				Server.data_buffer[0] := 1;
				Server.data_buffer[1] := TempSeqNum;
				Server.data_buffer[2] := LEN('Sequence Number Mismatch');
				brsmemcpy(ADR(Server.data_buffer[3]), ADR('Sequence Number Mismatch'),LEN('Sequence Number Mismatch'));
				Server.sStep := 30;

			ELSIF Server.TcpRecv_0.status = tcpERR_NO_DATA THEN  (* No data received - wait *)
			   Server.recv_timeout := Server.recv_timeout + 1;
			  IF Server.recv_timeout > 17500 THEN //Wait 35s
	 		    Server.sStep := 40;
				Server.recv_timeout := 0;
			  END_IF
			ELSIF Server.TcpRecv_0.status = ERR_FUB_BUSY THEN  (* TcpRecv not finished -> redo *)
			  (* Busy *)
			ELSIF Server.TcpRecv_0.status = tcpERR_NOT_CONNECTED THEN
				Server.sStep := 40;
			ELSE  (* Goto Error Step *)
				Server.sStep := 100;
			END_IF

		30:	(* Send Data back to Client *)
			prevStep := Server.sStep;
			Server.TcpSend_0.enable := 1;
			Server.TcpSend_0.ident := Server.TcpServer_0.identclnt;  (* Client Ident from AsTCP.TCP_Server *)
			Server.TcpSend_0.pData := ADR(Server.data_buffer[0]);  (* Which data to send *)
			IF Server.data_buffer[0] = 0 THEN
				Server.TcpSend_0.datalen := 8;  (* Lenght of data to send *)
			ELSE
				Server.TcpSend_0.datalen := 12 + Server.data_buffer[2];
			END_IF
			Server.TcpSend_0.flags := 0;
			Server.TcpSend_0;  (* Call the Function*)

			IF Server.TcpSend_0.status = 0 THEN  (* Data sent *)
				Server.sStep := 20;

			ELSIF Server.TcpSend_0.status = ERR_FUB_BUSY THEN  (* TcpSend not finished -> redo *)
			  (* Busy *)
			ELSIF (Server.TcpSend_0.status = tcpERR_NOT_CONNECTED) THEN
				Server.sStep := 40;
			ELSE  (* Goto Error Step *)
				Server.sStep := 100;
			END_IF

		40:
			prevStep := Server.sStep;
			Server.TcpClose_0.enable := 1;
			Server.TcpClose_0.ident := Server.TcpServer_0.identclnt;
			Server.TcpClose_0.how := 0; // tcpSHUT_RD OR tcpSHUT_WR;
			Server.TcpClose_0;

			IF Server.TcpClose_0.status = 0 THEN
   				Server.sStep := 50;
			ELSIF Server.TcpClose_0.status = ERR_FUB_BUSY THEN  (* TcpClose not finished -> redo *)
			  (* Busy *)
			ELSE  (* Goto Error Step *)
				Server.sStep := 100;
			END_IF
		50:
			prevStep := Server.sStep;
			Server.TcpClose_0.enable := 1;
			Server.TcpClose_0.ident := Server.TcpOpen_0.ident;
			Server.TcpClose_0.how := 0; //tcpSHUT_RD OR tcpSHUT_WR;
			Server.TcpClose_0;

			IF Server.TcpClose_0.status = 0 THEN
   				Server.sStep := 0;
			ELSIF Server.TcpClose_0.status = ERR_FUB_BUSY THEN  (* TcpClose not finished -> redo *)
			  (* Busy *)
			ELSE  (* Goto Error Step *)
				Server.sStep := 100;
			END_IF

		100: (* Error State. Wait 10s, reopen port and try again *)

			TON_Reopen.IN := TRUE;
			IF TON_Reopen.Q THEN
				Server.sStep := prevStep;
				TON_Reopen.IN := FALSE;
			END_IF

	END_CASE

	TON_Reopen();
	TON_MessageTimeout();

END_PROGRAM
```
